// TIA Portal V17 export
// export: Created 2025-03-10T13:12:58.3879354Z, ExportSetting WithDefaults, DisplayName Totally Integrated Automation Portal, DisplayVersion V17 Update 8, DisplayName TIA Portal Openness, DisplayVersion V17 Update 8, DisplayName TIA Portal Version Control Interface, DisplayVersion V17, DisplayName SINAMICS Startdrive Advanced, DisplayVersion V17 SP2, DisplayName SINAMICS Startdrive G110M, G120, G120C, G120D, G120P, G115D, DisplayVersion V17 SP2, DisplayName SINAMICS Startdrive G130, G150, S120, S150, SINAMICS MV, S210, DisplayVersion V17 SP2, DisplayName STEP 7 Professional, DisplayVersion V17 Update 8, DisplayName SINUMERIK ONE STEP 7 Toolbox, DisplayVersion V17 Update 12, DisplayName SINUMERIK 840D sl STEP 7 Toolbox, DisplayVersion V17 Update 12, DisplayName STEP 7 Safety, DisplayVersion V17 Update 6, DisplayName WinCC Advanced, DisplayVersion V17 Update 8
FUNCTION_BLOCK "FB22101_PRESSURE_SENSOR"   // FB22101, LAD
TITLE = FB22101 PRESSURE SENSOR
{ S7_Optimized_Access := 'FALSE' }
VERSION : 0.1
// stored: AutoNumber false, IsIECCheckEnabled false, SetENOAutomatically false, UDAEnableTagReadback false
   VAR_INPUT
      iINPUT_VALUE : Int;
      iCLEAR_INTERNAL_LOG : Bool;
      iSAVE_MAX_PRESSURE : Bool;
   END_VAR
   VAR_OUTPUT
      oWARNING_LIMIT : Bool;
      oERROR_LIMIT : Bool;
   END_VAR
   VAR DB_SPECIFIC
      OUTPUT : Struct
         VALUE : Real;
      END_STRUCT;
      INPUT_SETTINGS : Struct
         DIV_VALUE : Real := 1000.0;
         NORM_MIN_VALUE : DInt;
         NORM_MAX_VALUE : DInt := 27648;
         LOW_RANGE : Real;
         HIGH_RANGE : Real;
         IS_ANALOG_VALUE : Bool;
         UNIT_NUMBER : Int;
         HOPPER_NUMBER : Int;
      END_STRUCT;
      ALARMS_SETTINGS : Struct
         WARN_LIM_LOW : Real;
         ERROR_LIM_LOW : Real;
         WARN_LIM_HIGH : Real;
         ERROR_LIM_HIGH : Real;
         ERROR_CONFIGURATION : Bool;
      END_STRUCT;
      LOG : Struct
         DATE_MAX_PRESSURE : Date_And_Time;
         "VALUE_MAX PRESSURE" : Real;
      END_STRUCT;
      INTERNAL : Struct
         AUXILIARY_TRIGGER : Bool;
      END_STRUCT;
   END_VAR
   VAR_TEMP
      DB_NUMBER : DInt;
      RET_VAL : Int;
      ZERO : Int;
      NORM_VALUE : Real;
      CONV_VALUE : Real;
   END_VAR
   VAR_TEMP   // added for the SCL form of the ladder/FBD networks
      _w1 : Bool;
      _w2 : Bool;
   END_VAR
BEGIN

NETWORK
TITLE = READ INSTANCE DB NUMBER
      L     DINO;
      +     10#800000;
      T     #DB_NUMBER;

REGION Network 2: NORM AND SCALE ANALOG INPUT VALUE
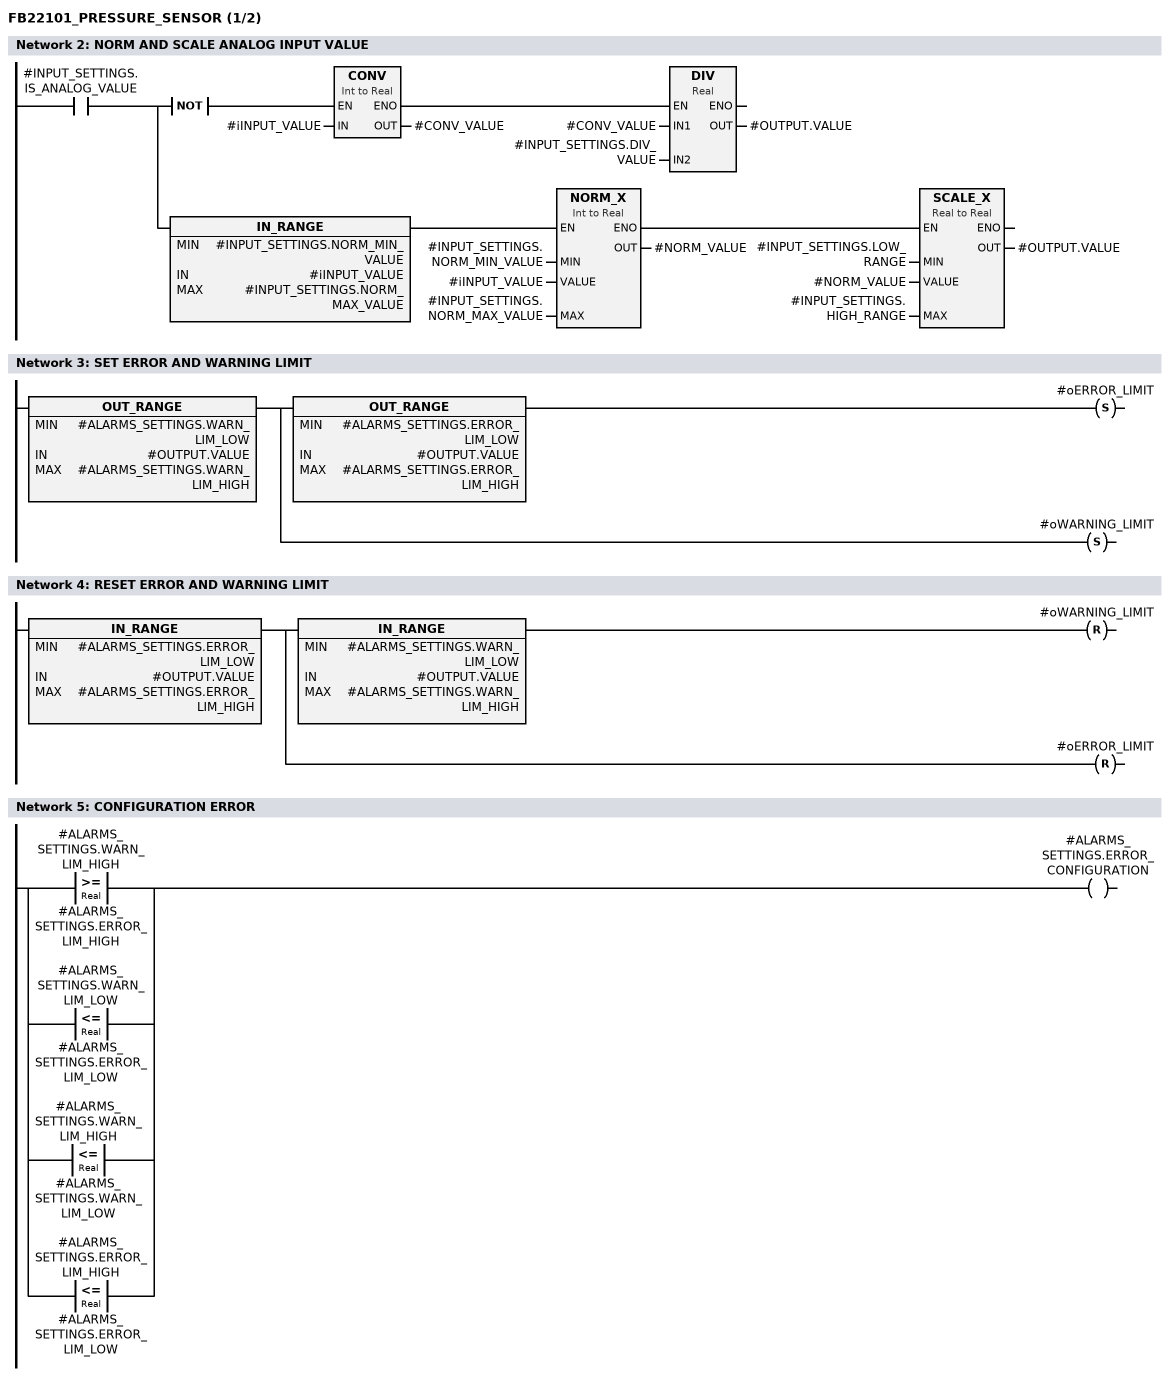
   RUNG wire#powerrail
      Contact( #INPUT_SETTINGS.IS_ANALOG_VALUE )
      wire#w1
      Not()
      { S7_Templates := "[SrcType := Int, DestType := Real]" } Convert(in := #iINPUT_VALUE, out => #CONV_VALUE)
      { S7_Templates := "SrcType := Real" } Div(in1 := #CONV_VALUE, in2 := #INPUT_SETTINGS.DIV_VALUE, out => #OUTPUT.VALUE)
   END_RUNG
   RUNG wire#w1
      { S7_Templates := "SrcType := DInt" } InRange(min := #INPUT_SETTINGS.NORM_MIN_VALUE, in := #iINPUT_VALUE, max := #INPUT_SETTINGS.NORM_MAX_VALUE)
      { S7_Templates := "[SrcType := Int, DestType := Real]" } Normalize(min := #INPUT_SETTINGS.NORM_MIN_VALUE, value := #iINPUT_VALUE, max := #INPUT_SETTINGS.NORM_MAX_VALUE, out => #NORM_VALUE)
      { S7_Templates := "[SrcType := Real, DestType := Real]" } Scale(min := #INPUT_SETTINGS.LOW_RANGE, value := #NORM_VALUE, max := #INPUT_SETTINGS.HIGH_RANGE, out => #OUTPUT.VALUE)
   END_RUNG
   // the same network as SCL:
   IF NOT #INPUT_SETTINGS.IS_ANALOG_VALUE THEN
       #CONV_VALUE := INT_TO_REAL(#iINPUT_VALUE);
       #OUTPUT.VALUE := #CONV_VALUE / #INPUT_SETTINGS.DIV_VALUE;
   END_IF;
   IF #INPUT_SETTINGS.IS_ANALOG_VALUE AND (#INPUT_SETTINGS.NORM_MIN_VALUE <= #iINPUT_VALUE) AND (#iINPUT_VALUE <= #INPUT_SETTINGS.NORM_MAX_VALUE) THEN
       #NORM_VALUE := NORM_X(MIN := #INPUT_SETTINGS.NORM_MIN_VALUE, VALUE := #iINPUT_VALUE, MAX := #INPUT_SETTINGS.NORM_MAX_VALUE);
       #OUTPUT.VALUE := SCALE_X(MIN := #INPUT_SETTINGS.LOW_RANGE, VALUE := #NORM_VALUE, MAX := #INPUT_SETTINGS.HIGH_RANGE);
   END_IF;
END_REGION

REGION Network 3: SET ERROR AND WARNING LIMIT
   #_w1 := (#OUTPUT.VALUE < #ALARMS_SETTINGS.WARN_LIM_LOW) OR (#OUTPUT.VALUE > #ALARMS_SETTINGS.WARN_LIM_HIGH);
   IF #_w1 AND ((#OUTPUT.VALUE < #ALARMS_SETTINGS.ERROR_LIM_LOW) OR (#OUTPUT.VALUE > #ALARMS_SETTINGS.ERROR_LIM_HIGH)) THEN
       #oERROR_LIMIT := TRUE;
   END_IF;
   IF #_w1 THEN #oWARNING_LIMIT := TRUE; END_IF;
END_REGION

REGION Network 4: RESET ERROR AND WARNING LIMIT
   RUNG wire#powerrail
      { S7_Templates := "SrcType := Real" } InRange(min := #ALARMS_SETTINGS.ERROR_LIM_LOW, in := #OUTPUT.VALUE, max := #ALARMS_SETTINGS.ERROR_LIM_HIGH)
      wire#w1
      { S7_Templates := "SrcType := Real" } InRange(min := #ALARMS_SETTINGS.WARN_LIM_LOW, in := #OUTPUT.VALUE, max := #ALARMS_SETTINGS.WARN_LIM_HIGH)
      R_Coil( #oWARNING_LIMIT )
   END_RUNG
   RUNG wire#w1
      R_Coil( #oERROR_LIMIT )
   END_RUNG
   // the same network as SCL:
   #_w1 := (#ALARMS_SETTINGS.ERROR_LIM_LOW <= #OUTPUT.VALUE) AND (#OUTPUT.VALUE <= #ALARMS_SETTINGS.ERROR_LIM_HIGH);
   IF #_w1 AND (#ALARMS_SETTINGS.WARN_LIM_LOW <= #OUTPUT.VALUE) AND (#OUTPUT.VALUE <= #ALARMS_SETTINGS.WARN_LIM_HIGH) THEN
       #oWARNING_LIMIT := FALSE;
   END_IF;
   IF #_w1 THEN #oERROR_LIMIT := FALSE; END_IF;
END_REGION

REGION Network 5: CONFIGURATION ERROR
   RUNG wire#powerrail
      { S7_Templates := "SrcType := Real" } GE_Contact(in1 := #ALARMS_SETTINGS.WARN_LIM_HIGH, in2 := #ALARMS_SETTINGS.ERROR_LIM_HIGH)
      wire#w1
      Coil( #ALARMS_SETTINGS.ERROR_CONFIGURATION )
   END_RUNG
   RUNG wire#powerrail
      { S7_Templates := "SrcType := Real" } LE_Contact(in1 := #ALARMS_SETTINGS.WARN_LIM_LOW, in2 := #ALARMS_SETTINGS.ERROR_LIM_LOW)
   END_RUNG wire#w1
   RUNG wire#powerrail
      { S7_Templates := "SrcType := Real" } LE_Contact(in1 := #ALARMS_SETTINGS.WARN_LIM_HIGH, in2 := #ALARMS_SETTINGS.WARN_LIM_LOW)
   END_RUNG wire#w1
   RUNG wire#powerrail
      { S7_Templates := "SrcType := Real" } LE_Contact(in1 := #ALARMS_SETTINGS.ERROR_LIM_HIGH, in2 := #ALARMS_SETTINGS.ERROR_LIM_LOW)
   END_RUNG wire#w1
   // the same network as SCL:
   #ALARMS_SETTINGS.ERROR_CONFIGURATION := (#ALARMS_SETTINGS.WARN_LIM_HIGH >= #ALARMS_SETTINGS.ERROR_LIM_HIGH) OR (#ALARMS_SETTINGS.WARN_LIM_LOW <= #ALARMS_SETTINGS.ERROR_LIM_LOW) OR (#ALARMS_SETTINGS.WARN_LIM_HIGH <= #ALARMS_SETTINGS.WARN_LIM_LOW) OR (#ALARMS_SETTINGS.ERROR_LIM_HIGH <= #ALARMS_SETTINGS.ERROR_LIM_LOW);
END_REGION

REGION Network 6: SAVE MAX PRESSURE
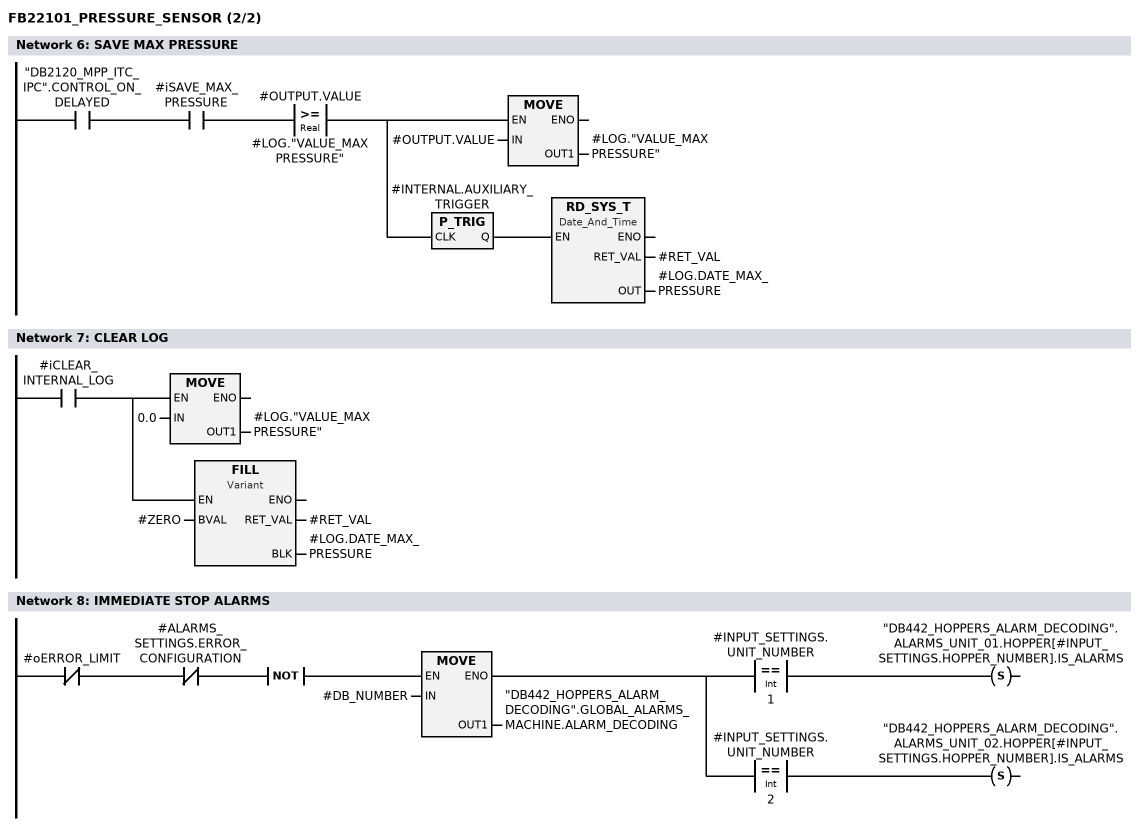
   RUNG wire#powerrail
      Contact( "DB2120_MPP_ITC_IPC".CONTROL_ON_DELAYED )
      Contact( #iSAVE_MAX_PRESSURE )
      { S7_Templates := "SrcType := Real" } GE_Contact(in1 := #OUTPUT.VALUE, in2 := #LOG."VALUE_MAX PRESSURE")
      wire#w1
      Move(in := #OUTPUT.VALUE, out1 => #LOG."VALUE_MAX PRESSURE")
   END_RUNG
   RUNG wire#w1
      P_Trig( #INTERNAL.AUXILIARY_TRIGGER )
      { S7_Templates := "date_type := Date_And_Time" } RD_SYS_T(RET_VAL => #RET_VAL, OUT => #LOG.DATE_MAX_PRESSURE)
   END_RUNG
   // the same network as SCL:
   #_w1 := "DB2120_MPP_ITC_IPC".CONTROL_ON_DELAYED AND #iSAVE_MAX_PRESSURE AND (#OUTPUT.VALUE >= #LOG."VALUE_MAX PRESSURE");
   IF #_w1 THEN #LOG."VALUE_MAX PRESSURE" := #OUTPUT.VALUE; END_IF;
   #_w2 := #_w1 AND NOT #INTERNAL.AUXILIARY_TRIGGER;   // rising edge
   #INTERNAL.AUXILIARY_TRIGGER := #_w1;
   IF #_w2 THEN #RET_VAL := RD_SYS_T(OUT => #LOG.DATE_MAX_PRESSURE); END_IF;
END_REGION

REGION Network 7: CLEAR LOG
   RUNG wire#powerrail
      Contact( #iCLEAR_INTERNAL_LOG )
      wire#w1
      { S7_GenerateENO := "TRUE" } Move(in := 0.0, out1 => #LOG."VALUE_MAX PRESSURE")
   END_RUNG
   RUNG wire#w1
      { S7_Templates := "ptr_type := Variant" } FILL(BVAL := #ZERO, RET_VAL => #RET_VAL, BLK => #LOG.DATE_MAX_PRESSURE)
   END_RUNG
   // the same network as SCL:
   IF #iCLEAR_INTERNAL_LOG THEN
       #LOG."VALUE_MAX PRESSURE" := 0.0;
       #RET_VAL := FILL(BVAL := #ZERO, BLK => #LOG.DATE_MAX_PRESSURE);
   END_IF;
END_REGION

REGION Network 8: IMMEDIATE STOP ALARMS
   RUNG wire#powerrail
      I_Contact( #oERROR_LIMIT )
      I_Contact( #ALARMS_SETTINGS.ERROR_CONFIGURATION )
      Not()
      { S7_GenerateENO := "TRUE" } Move(in := #DB_NUMBER, out1 => "DB442_HOPPERS_ALARM_DECODING".GLOBAL_ALARMS_MACHINE.ALARM_DECODING)
      wire#w1
      { S7_Templates := "SrcType := Int" } EQ_Contact(in1 := #INPUT_SETTINGS.UNIT_NUMBER, in2 := 1)
      S_Coil( "DB442_HOPPERS_ALARM_DECODING".ALARMS_UNIT_01.HOPPER[#INPUT_SETTINGS.HOPPER_NUMBER].IS_ALARMS )
   END_RUNG
   RUNG wire#w1
      { S7_Templates := "SrcType := Int" } EQ_Contact(in1 := #INPUT_SETTINGS.UNIT_NUMBER, in2 := 2)
      S_Coil( "DB442_HOPPERS_ALARM_DECODING".ALARMS_UNIT_02.HOPPER[#INPUT_SETTINGS.HOPPER_NUMBER].IS_ALARMS )
   END_RUNG
   // the same network as SCL:
   // ENO of a box is taken as its EN; it also drops when the box reports an error
   #_w1 := NOT (NOT #oERROR_LIMIT AND NOT #ALARMS_SETTINGS.ERROR_CONFIGURATION);
   IF #_w1 THEN "DB442_HOPPERS_ALARM_DECODING".GLOBAL_ALARMS_MACHINE.ALARM_DECODING := #DB_NUMBER; END_IF;
   IF #_w1 AND (#INPUT_SETTINGS.UNIT_NUMBER = 1) THEN
       "DB442_HOPPERS_ALARM_DECODING".ALARMS_UNIT_01.HOPPER[#INPUT_SETTINGS.HOPPER_NUMBER].IS_ALARMS := TRUE;
   END_IF;
   IF #_w1 AND (#INPUT_SETTINGS.UNIT_NUMBER = 2) THEN
       "DB442_HOPPERS_ALARM_DECODING".ALARMS_UNIT_02.HOPPER[#INPUT_SETTINGS.HOPPER_NUMBER].IS_ALARMS := TRUE;
   END_IF;
END_REGION
END_FUNCTION_BLOCK
